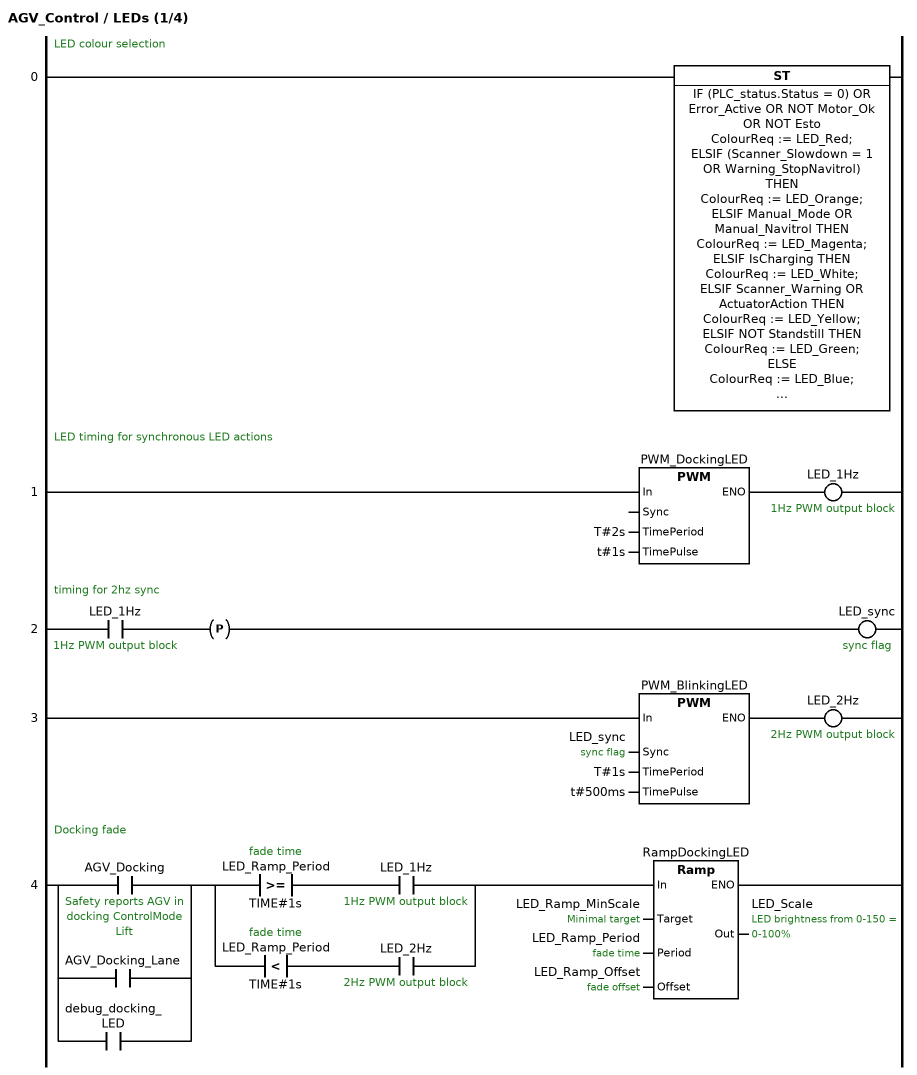
(* [picture p19: AGV_Control / LEDs, rungs 0-4] *)
(* Rung 0: LED colour selection *)
IF (PLC_status.Status = 0) OR Error_Active OR NOT Motor_Ok OR NOT Estop_Out OR (Warning_Mqtt_Client_Error AND InProd) THEN
	ColourReq := LED_Red;
ELSIF (Scanner_Slowdown = 1 OR Warning_StopNavitrol) THEN
	ColourReq := LED_Orange;
ELSIF Manual_Mode OR Manual_Navitrol THEN
	ColourReq := LED_Magenta;
ELSIF IsCharging THEN
	ColourReq := LED_White;
ELSIF Scanner_Warning OR ActuatorAction THEN
	ColourReq := LED_Yellow;
ELSIF NOT Standstill THEN
	ColourReq := LED_Green;
ELSE
	ColourReq := LED_Blue;
END_IF;

IF NOT debug_LED THEN
	Colour := ColourReq;
ELSE
	Colour := debug_Colour;
END_IF;

CASE Colour OF
	LED_Red:
		LED_R_Req := 100;
		LED_G_Req := 0;
		LED_B_Req := 0;
	LED_Orange:
		LED_R_Req := 100;
		LED_G_Req := 50;
		LED_B_Req := 0;
	LED_Yellow:
		LED_R_Req := 75;
		LED_G_Req := 75;
		LED_B_Req := 0;
	LED_Green:
		LED_R_Req := 0;
		LED_G_Req := 100;
		LED_B_Req := 0;
	LED_Cyan:
		LED_R_Req := 0;
		LED_G_Req := 100;
		LED_B_Req := 100;
	LED_Blue:
		LED_R_Req := 0;
		LED_G_Req := 0;
		LED_B_Req := 100;
	LED_Magenta:
		LED_R_Req := 100;
		LED_G_Req := 0;
		LED_B_Req := 100;
	LED_White:
		LED_R_Req := 100;
		LED_G_Req := 100;
		LED_B_Req := 100;
END_CASE;

IF (Colour = LED_Colour#LED_Orange) THEN
	LED_R := LED_R_Req*LED_Scale;
	LED_G := LED_G_Req*LED_Scale;//REAL_TO_INT(LED_R / 2) + ((LED_Ramp_Offset-LED_Scale) * 8);
	LED_B := LED_B_Req*LED_Scale;
ELSE
	LED_R := LED_R_Req*LED_Scale;
	LED_G := LED_G_Req*LED_Scale;
	LED_B := LED_B_Req*LED_Scale;
END_IF;

IF DomeLEDs THEN
	 if( LED_R>0) AND (Colour <> LED_Colour#LED_Orange) THEN 
		 IF NOT AGV_Docking THEN
		 	O_LED_R := TRUE; 
		ELSE 
			O_LED_R := LED_1Hz;
		END_IF;
	 ELSE
		 O_LED_R := FALSE;
	 END_IF;
	 
	 if( LED_G>0)  THEN 
		 IF NOT AGV_Docking THEN
		 	O_LED_G := TRUE; 
		ELSE 
			O_LED_G := LED_1Hz;
		END_IF;
	 ELSE
		 O_LED_G := FALSE;
	 END_IF;

	 if( LED_B>0) OR (Colour = LED_Colour#LED_Orange) THEN 
		 IF NOT AGV_Docking THEN
		 	O_LED_B := TRUE; 
		ELSE 
			O_LED_B := LED_1Hz;
		END_IF;
	 ELSE
		 O_LED_B := FALSE;
	 END_IF;
END_IF;

IF (LED_Scale < 0) THEN
	LED_Scale := 0;
END_IF;
IF IsCharging OR NOT (AGV_Docking OR debug_docking_LED) THEN
	LED_Scale:= LED_Ramp_Offset;
END_IF;

isCharging := Charge_Relay AND Navitrol_Battery.Voltage > 267;
(* Rung 1: LED timing for synchronous LED actions *)
PWM_DockingLED(In := TRUE, TimePeriod := T#2s, TimePulse := t#1s);
LED_1Hz := PWM_DockingLED.ENO;
(* Rung 2: timing for 2hz sync *)
_e36(CLK := LED_1Hz);
LED_sync := _e36.Q;
(* Rung 3 *)
PWM_BlinkingLED(In := TRUE, Sync := LED_sync, TimePeriod := T#1s, TimePulse := t#500ms);
LED_2Hz := PWM_BlinkingLED.ENO;
(* Rung 4: Docking fade *)
RampDockingLED(In := (AGV_Docking OR AGV_Docking_Lane OR debug_docking_LED) AND (((LED_Ramp_Period >= TIME#1s) AND LED_1Hz) OR ((LED_Ramp_Period < TIME#1s) AND LED_2Hz)), Target := LED_Ramp_MinScale, Period := LED_Ramp_Period, Offset := LED_Ramp_Offset, Out => LED_Scale);

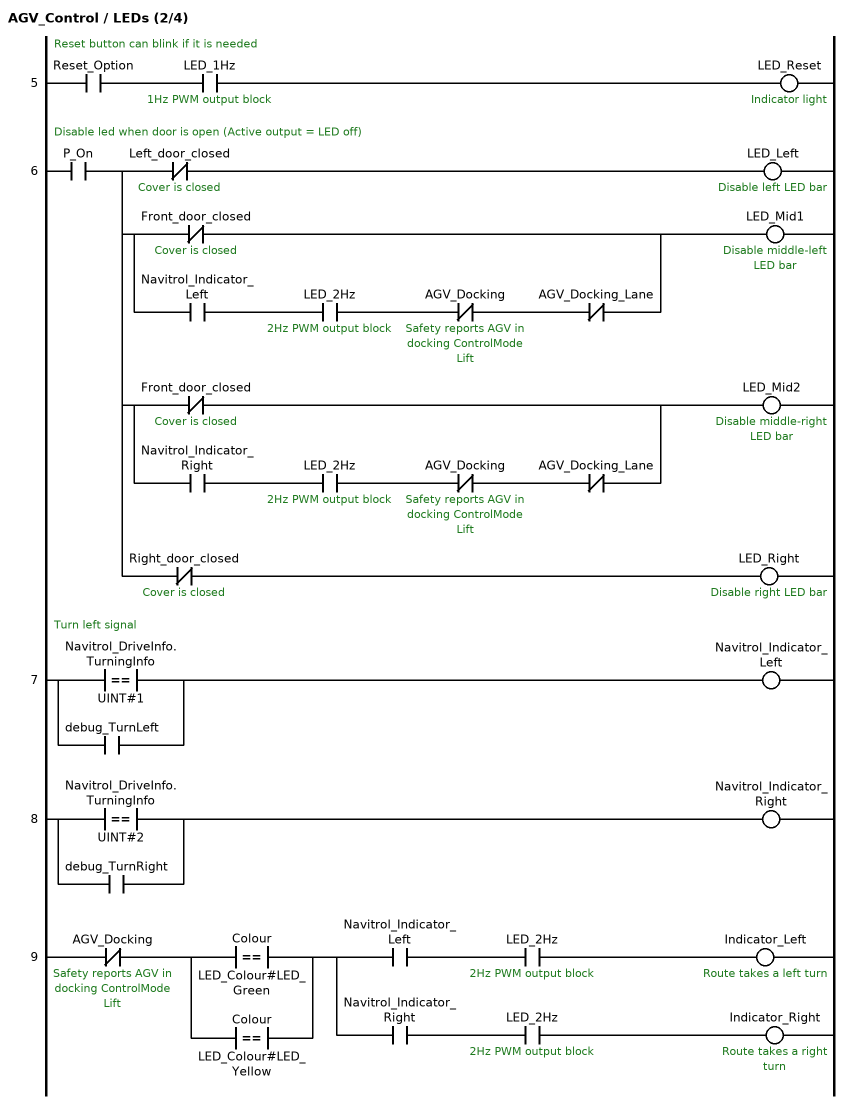
(* Rung 5: Reset button can blink if it is needed *)
LED_Reset := Reset_Option AND LED_1Hz;
(* Rung 6: Disable led when door is open (Active output = LED off) *)
LED_Left := P_On AND NOT Left_door_closed;
LED_Mid1 := P_On AND (NOT Front_door_closed OR (Navitrol_Indicator_Left AND LED_2Hz AND NOT AGV_Docking AND NOT AGV_Docking_Lane));
LED_Mid2 := P_On AND (NOT Front_door_closed OR (Navitrol_Indicator_Right AND LED_2Hz AND NOT AGV_Docking AND NOT AGV_Docking_Lane));
LED_Right := P_On AND NOT Right_door_closed;
(* Rung 7: Turn left signal *)
Navitrol_Indicator_Left := (Navitrol_DriveInfo.TurningInfo = UINT#1) OR debug_TurnLeft;
(* Rung 8 *)
Navitrol_Indicator_Right := (Navitrol_DriveInfo.TurningInfo = UINT#2) OR debug_TurnRight;
(* Rung 9 *)
_p37 := NOT AGV_Docking AND ((Colour = LED_Colour#LED_Green) OR (Colour = LED_Colour#LED_Yellow));
Indicator_Left := _p37 AND Navitrol_Indicator_Left AND LED_2Hz;
Indicator_Right := _p37 AND Navitrol_Indicator_Right AND LED_2Hz;

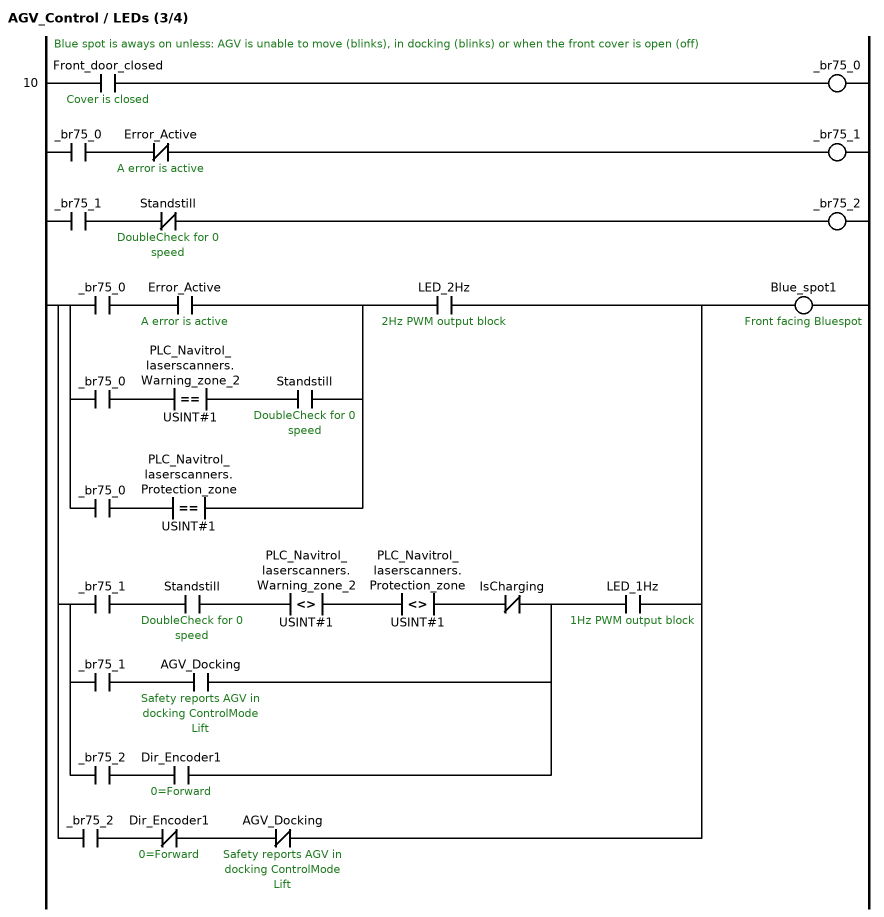
(* Rung 10: Blue spot is aways on unless: AGV is unable to move (blinks), in docking (blinks) or when the front cover is open (off) *)
_br75_0 := Front_door_closed;
_br75_1 := _br75_0 AND NOT Error_Active;
_br75_2 := _br75_1 AND NOT Standstill;
Blue_spot1 := (((_br75_0 AND Error_Active) OR (_br75_0 AND (PLC_Navitrol_laserscanners.Warning_zone_2 = USINT#1) AND Standstill) OR (_br75_0 AND (PLC_Navitrol_laserscanners.Protection_zone = USINT#1))) AND LED_2Hz) OR (((_br75_1 AND Standstill AND (PLC_Navitrol_laserscanners.Warning_zone_2 <> USINT#1) AND (PLC_Navitrol_laserscanners.Protection_zone <> USINT#1) AND NOT IsCharging) OR (_br75_1 AND AGV_Docking) OR (_br75_2 AND Dir_Encoder1)) AND LED_1Hz) OR (_br75_2 AND NOT Dir_Encoder1 AND NOT AGV_Docking);

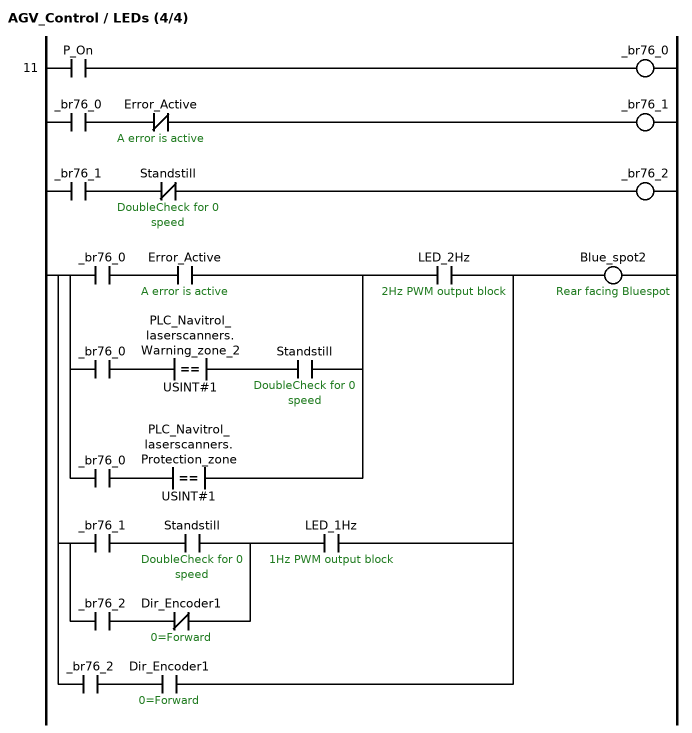
(* Rung 11 *)
_br76_0 := P_On;
_br76_1 := _br76_0 AND NOT Error_Active;
_br76_2 := _br76_1 AND NOT Standstill;
Blue_spot2 := (((_br76_0 AND Error_Active) OR (_br76_0 AND (PLC_Navitrol_laserscanners.Warning_zone_2 = USINT#1) AND Standstill) OR (_br76_0 AND (PLC_Navitrol_laserscanners.Protection_zone = USINT#1))) AND LED_2Hz) OR (((_br76_1 AND Standstill) OR (_br76_2 AND NOT Dir_Encoder1)) AND LED_1Hz) OR (_br76_2 AND Dir_Encoder1);

(* Section MES: ladder, written here as Structured Text *)

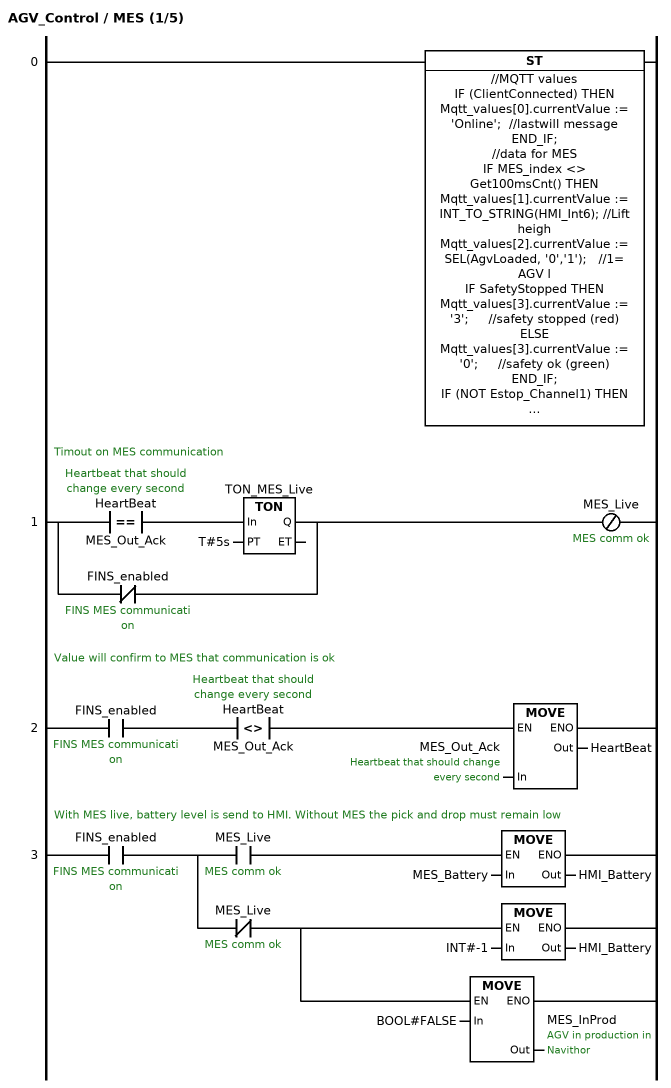
(* Rung 0 *)
//MQTT values
IF (ClientConnected) THEN
	Mqtt_values[0].currentValue := 'Online';	//lastwill message
END_IF;
//data for MES
IF MES_index <> Get100msCnt() THEN
	Mqtt_values[1].currentValue := INT_TO_STRING(HMI_Int6);	//Lift height in mm
	Mqtt_values[2].currentValue := SEL(AgvLoaded, '0','1');		//1= AGV loaded
	IF SafetyStopped THEN
	    Mqtt_values[3].currentValue := '3';			//safety stopped (red)
	ELSE
	    Mqtt_values[3].currentValue := '0';			//safety ok (green)
	END_IF;
	IF (NOT Estop_Channel1) THEN
		Mqtt_values[4].currentValue := '3';			//Estop button pressed (red)
	ELSIF (NOT Estop_Out) THEN
		Mqtt_values[4].currentValue := '2';			//Estop button ok, but not reset (yellow)
	ELSE
		Mqtt_values[4].currentValue := '0';			//Estop button ok (green)
	END_IF;
	Mqtt_values[5].currentValue := DINT_TO_STRING (EnumToNum(Scanner1_State));	//scanner status
	Mqtt_values[6].currentValue := DINT_TO_STRING (EnumToNum(Scanner2_State));	//scanner status
	Mqtt_values[7].currentValue := DINT_TO_STRING (EnumToNum(Scanner3_State));	//scanner status
	Mqtt_values[8].currentValue := SEL (OptionalFieldReq = 0,'1','0');	//1= Docking field active
	Mqtt_values[9].currentValue := SEL (Manual_Navitrol,'0','1');		//1= AGV in manualControlModeLift (navitrol)
	Mqtt_values[10].currentValue := SEL (HMI_Input5,'0','1');			//1= Lift in manual ControlModeLift
	Mqtt_values[11].currentValue := SEL (Brake_release,'0','1');	//1= Lift manually released
	Mqtt_values[12].currentValue := SEL (HMI_Int10 = 0,'0','1');	//1= AGV charging
	Mqtt_values[13].currentValue := SEL (MES_Request_Cancel, '0','1');	//1= MES can cancel order while AGV lowers fork
	IF (HMI_Int6 < 100 AND Mqtt_values[14].currentValue = '1' AND MES_Request_Cancel) OR Mqtt_values[14].currentValue = '' THEN
		Mqtt_values[14].currentValue := '0';	//order cancel completed, reset value
	END_IF;
	Mqtt_values[15].currentValue := SEL(Error_Fork_Object,'0','1');
	Mqtt_values[16].currentValue := INT_TO_STRING (CountedPallets);	//1= MES can cancel order while AGV lowers fork

	Mqtt_values[17].currentValue := SEL (lift_heavyLoad,'0','1');	//1 = There is heavy load on the forks
	Mqtt_values[18].currentValue := DINT_TO_STRING (EnumToNum(MES_LaneDropState)); // Lane drop state
	Mqtt_values[22].currentValue := SEL (HMI_Input11,'0','1');	//1= The question for certain action is answered with "Yes"
	Mqtt_values[23].currentValue := SEL (HMI_Input12,'0','1');	//1= The question for certain action is answered with "Cancel"
	Mqtt_values[24].currentValue := INT_TO_STRING(MES_Language);
	Mqtt_values[25].currentValue := DINT_TO_STRING (EnumToNum(MES_LanePickState)); // Lane drop state
	
	Navitrol_TargetDetectionStatusToMES.TargetFount := SEL	(Navitrol_TargetDetectionStatus.TargetFount= 01, '0,','1,'); 
	Navitrol_TargetDetectionStatusToMES.TargetReached := SEL	(Navitrol_TargetDetectionStatus.TargetReached= 01, '0,','1,'); 	
	Navitrol_TargetDetectionStatusToMES.TargetWithinSafetyDistance := SEL  (Navitrol_TargetDetectionStatus.TargetWithinSafetyDistance = 01, '0,','1,'); 	
	Navitrol_TargetDetectionStatusToMES.TargetX := 	(INT_TO_STRING (REAL_TO_INT (Navitrol_TargetDetectionStatus.TargetX*100 ))); 
	Navitrol_TargetDetectionStatusToMES.TargetY := (INT_TO_STRING (REAL_TO_INT 	(Navitrol_TargetDetectionStatus.TargetY*100))); 	
	Navitrol_TargetDetectionStatusToMES.Angle:= (INT_TO_STRING (REAL_TO_INT 	(Navitrol_TargetDetectionStatus.TargetAngle*100))); 
	
	Mqtt_values[19].currentValue :=CONCAT (Navitrol_TargetDetectionStatusToMES.TargetFount,Navitrol_TargetDetectionStatusToMES.TargetReached,
	Navitrol_TargetDetectionStatusToMES.TargetWithinSafetyDistance,CONCAT (Navitrol_TargetDetectionStatusToMES.TargetX,','),Navitrol_TargetDetectionStatusToMES.TargetY);

	Mqtt_values[21].currentValue :=Navitrol_TargetDetectionStatusToMES.Angle;
	//error list to MES
	IF Navitrol_ErrorWithLevel.ErrorCount = 0 THEN
		//no error, clear values
		Mqtt_values[20].currentValue := '';
	ELSE
		ErrorString := '';
		FOR index := 0 TO UDINT_TO_INT(Navitrol_ErrorWithLevel.ErrorCount)-1 DO
			ErrorString := CONCAT(ErrorString, UDINT_TO_STRING(Navitrol_ErrorWithLevel.ErrorList[index].ErrorCode),',');
		END_FOR;
		Mqtt_values[20].currentValue := ErrorString;
	END_IF;
	
	MES_index := Get100msCnt();
END_IF;
//MQTT actuator request
(* Rung 1: Timout on MES communication *)
TON_MES_Live(In := HeartBeat = MES_Out_Ack, PT := T#5s);
MES_Live := NOT (TON_MES_Live.Q OR NOT FINS_enabled);
(* Rung 2: Value will confirm to MES that communication is ok *)
IF FINS_enabled AND (HeartBeat <> MES_Out_Ack) THEN HeartBeat := MES_Out_Ack; END_IF;
(* Rung 3: With MES live, battery level is send to HMI. Without MES the pick and drop must remain low *)
IF FINS_enabled AND MES_Live THEN HMI_Battery := MES_Battery; END_IF;
IF FINS_enabled AND NOT MES_Live THEN
    HMI_Battery := INT#-1;
    MES_InProd := BOOL#FALSE;
END_IF;

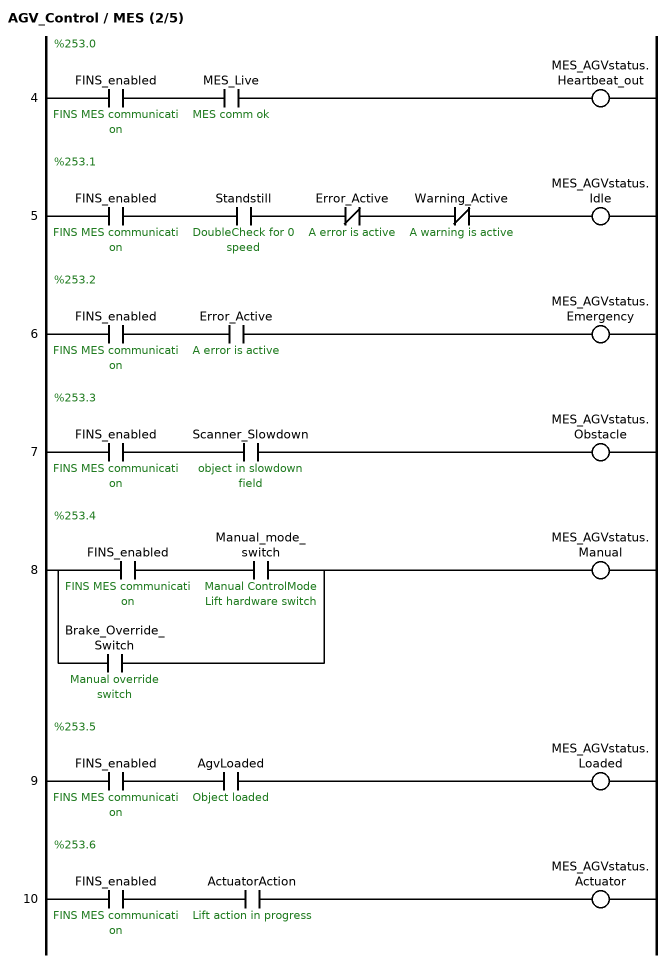
(* Rung 4: %253.0 *)
MES_AGVstatus.Heartbeat_out := FINS_enabled AND MES_Live;
(* Rung 5: %253.1 *)
MES_AGVstatus.Idle := FINS_enabled AND Standstill AND NOT Error_Active AND NOT Warning_Active;
(* Rung 6: %253.2 *)
MES_AGVstatus.Emergency := FINS_enabled AND Error_Active;
(* Rung 7: %253.3 *)
MES_AGVstatus.Obstacle := FINS_enabled AND Scanner_Slowdown;
(* Rung 8: %253.4 *)
MES_AGVstatus.Manual := (FINS_enabled AND Manual_mode_switch) OR Brake_Override_Switch;
(* Rung 9: %253.5 *)
MES_AGVstatus.Loaded := FINS_enabled AND AgvLoaded;
(* Rung 10: %253.6 *)
MES_AGVstatus.Actuator := FINS_enabled AND ActuatorAction;

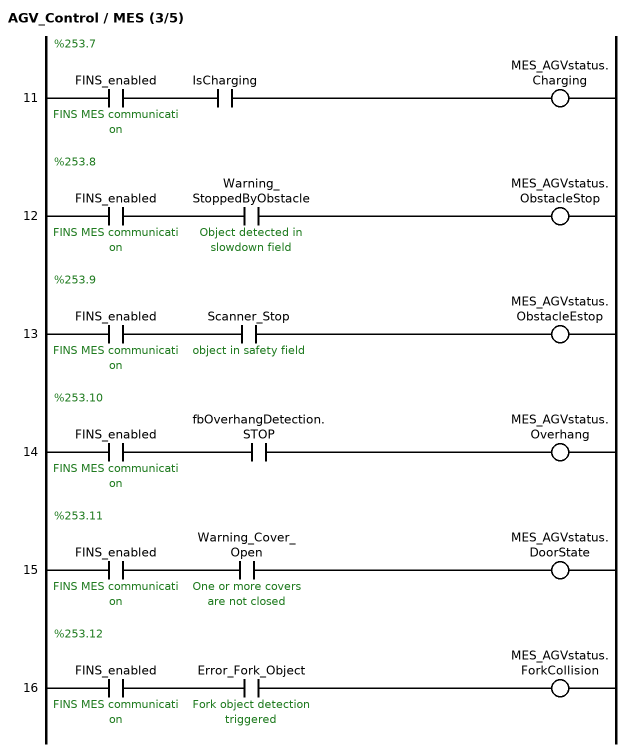
(* Rung 11: %253.7 *)
MES_AGVstatus.Charging := FINS_enabled AND IsCharging;
(* Rung 12: %253.8 *)
MES_AGVstatus.ObstacleStop := FINS_enabled AND Warning_StoppedByObstacle;
(* Rung 13: %253.9 *)
MES_AGVstatus.ObstacleEstop := FINS_enabled AND Scanner_Stop;
(* Rung 14: %253.10 *)
MES_AGVstatus.Overhang := FINS_enabled AND fbOverhangDetection.STOP;
(* Rung 15: %253.11 *)
MES_AGVstatus.DoorState := FINS_enabled AND Warning_Cover_Open;
(* Rung 16: %253.12 *)
MES_AGVstatus.ForkCollision := FINS_enabled AND Error_Fork_Object;

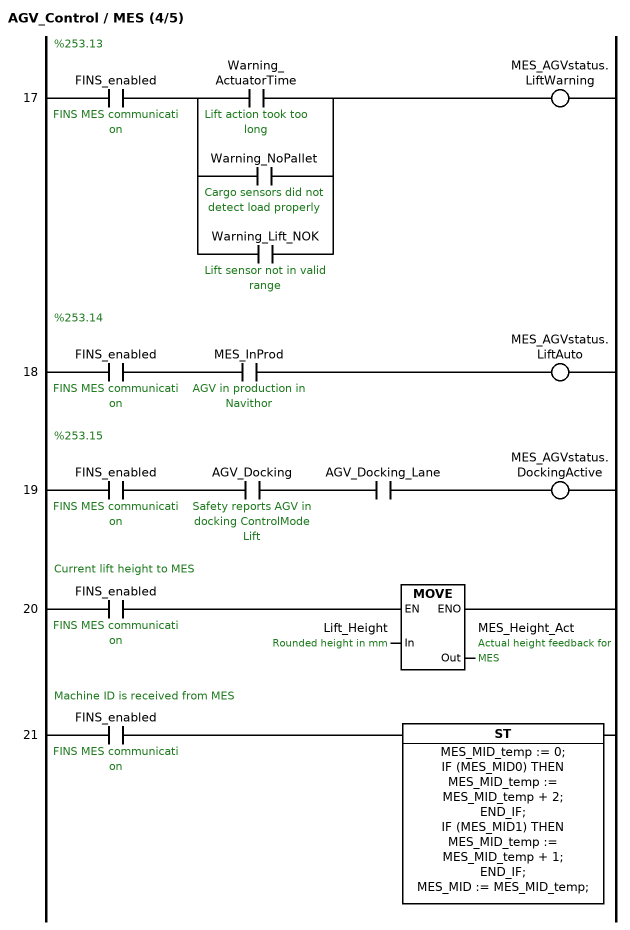
(* Rung 17: %253.13 *)
MES_AGVstatus.LiftWarning := FINS_enabled AND (Warning_ActuatorTime OR Warning_NoPallet OR Warning_Lift_NOK);
(* Rung 18: %253.14 *)
MES_AGVstatus.LiftAuto := FINS_enabled AND MES_InProd;
(* Rung 19: %253.15 *)
MES_AGVstatus.DockingActive := FINS_enabled AND AGV_Docking AND AGV_Docking_Lane;
(* Rung 20: Current lift height to MES *)
IF FINS_enabled THEN MES_Height_Act := Lift_Height; END_IF;
(* Rung 21: Machine ID is received from MES *)
IF FINS_enabled THEN
    MES_MID_temp := 0;
    IF (MES_MID0) THEN
    	MES_MID_temp := MES_MID_temp + 2;
    END_IF;
    IF (MES_MID1) THEN
    	MES_MID_temp := MES_MID_temp + 1;
    END_IF;
    MES_MID := MES_MID_temp;
END_IF;

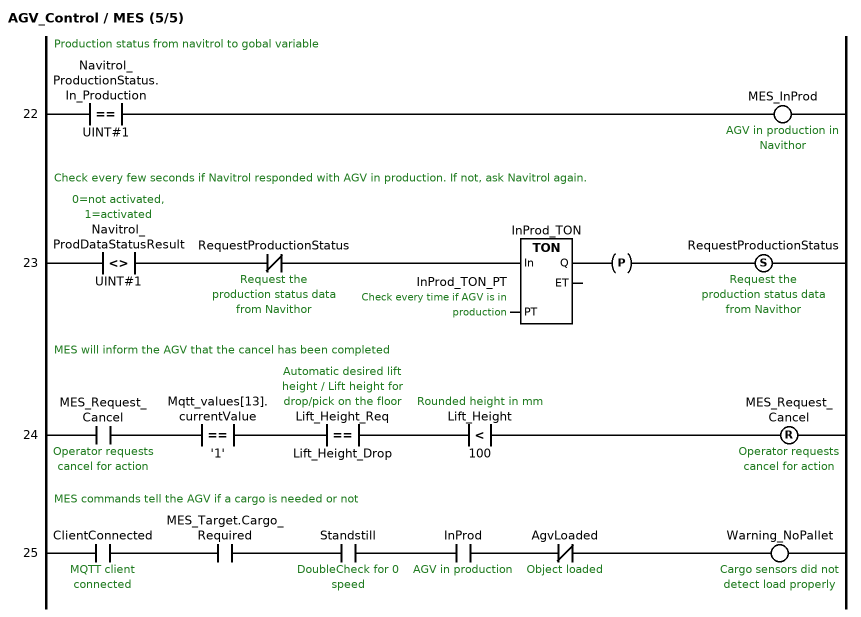
(* Rung 22: Production status from navitrol to gobal variable *)
MES_InProd := Navitrol_ProductionStatus.In_Production = UINT#1;
(* Rung 23: Check every few seconds if Navitrol responded with AGV in production. If not, ask Navitrol again. *)
InProd_TON(In := (Navitrol_ProdDataStatusResult <> UINT#1) AND NOT RequestProductionStatus, PT := InProd_TON_PT);
_e38(CLK := InProd_TON.Q);
IF _e38.Q THEN RequestProductionStatus := TRUE; END_IF;
(* Rung 24: MES will inform the AGV that the cancel has been completed *)
IF MES_Request_Cancel AND (Mqtt_values[13].currentValue = '1') AND (Lift_Height_Req = Lift_Height_Drop) AND (Lift_Height < 100) THEN
    MES_Request_Cancel := FALSE;
END_IF;
(* Rung 25: MES commands tell the AGV if a cargo is needed or not *)
Warning_NoPallet := ClientConnected AND MES_Target.Cargo_Required AND Standstill AND InProd AND NOT AgvLoaded;

(* Section HMI: ladder, written here as Structured Text *)

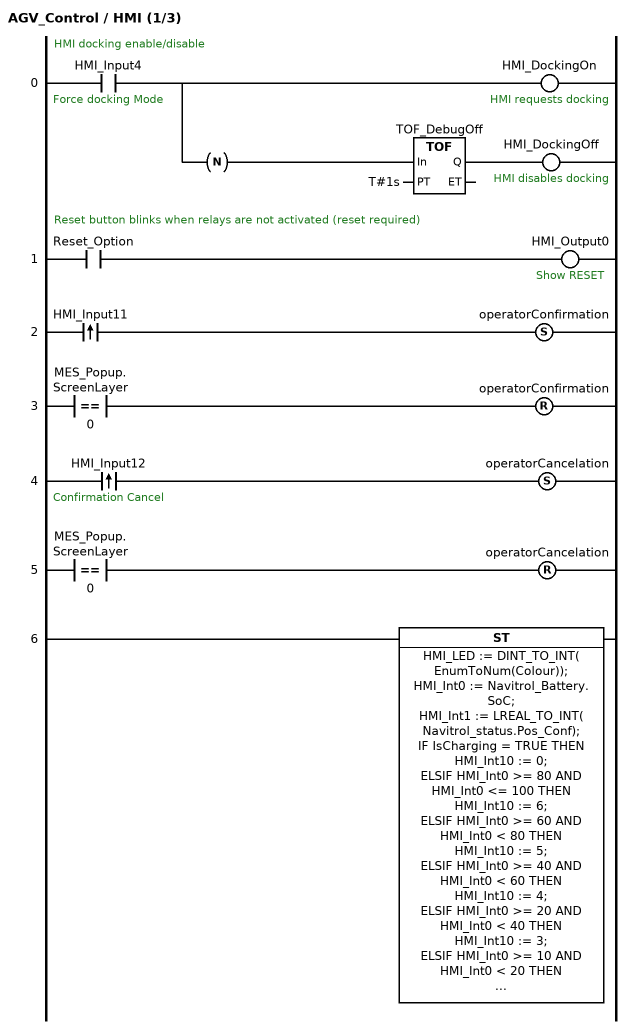
(* Rung 0: HMI docking enable/disable *)
HMI_DockingOn := HMI_Input4;
_e39(CLK := HMI_Input4);
TOF_DebugOff(In := _e39.Q, PT := T#1s);
HMI_DockingOff := TOF_DebugOff.Q;
(* Rung 1: Reset button blinks when relays are not activated (reset required) *)
HMI_Output0 := Reset_Option;
(* Rung 2 *)
_e40(CLK := HMI_Input11);
IF _e40.Q THEN operatorConfirmation := TRUE; END_IF;
(* Rung 3 *)
IF MES_Popup.ScreenLayer = 0 THEN operatorConfirmation := FALSE; END_IF;
(* Rung 4 *)
_e41(CLK := HMI_Input12);
IF _e41.Q THEN operatorCancelation := TRUE; END_IF;
(* Rung 5 *)
IF MES_Popup.ScreenLayer = 0 THEN operatorCancelation := FALSE; END_IF;
(* Rung 6 *)
HMI_LED := DINT_TO_INT(EnumToNum(Colour));

HMI_Int0 := Navitrol_Battery.SoC;
HMI_Int1 := LREAL_TO_INT(Navitrol_status.Pos_Conf);

IF IsCharging = TRUE THEN
	HMI_Int10 := 0;
ELSIF HMI_Int0 >= 80 AND HMI_Int0 <= 100 THEN
	HMI_Int10 := 6;
ELSIF HMI_Int0 >= 60 AND HMI_Int0 < 80 THEN
	HMI_Int10 := 5;
ELSIF HMI_Int0 >= 40 AND HMI_Int0 < 60 THEN
	HMI_Int10 := 4;
ELSIF HMI_Int0 >= 20 AND HMI_Int0 < 40 THEN
	HMI_Int10 := 3;
ELSIF HMI_Int0 >= 10 AND HMI_Int0 < 20 THEN
	HMI_Int10 := 2;
ELSE  //HMI_Int0 < 10 & not charging
	HMI_Int10 := 1;
END_IF;

//front scanners cmbined till HMI is updated
IF NOT Scan1_Stop OR NOT Scan2_Stop THEN
	Scanner1_State := State_Scanner#SCAN_eStop;
	Scanner2_State := State_Scanner#SCAN_eStop;
	HMI_Int2 := 0;
ELSIF NOT Scan1_Slow OR NOT Scan2_Slow THEN
	Scanner1_State := State_Scanner#SCAN_Stop;
	Scanner2_State := State_Scanner#SCAN_Stop;
	HMI_Int2 := 3;
ELSIF NOT Scan1_Warn OR NOT Scan2_Warn THEN
	Scanner1_State := State_Scanner#SCAN_Warn;
	Scanner2_State := State_Scanner#SCAN_Warn;
	HMI_Int2 := 2;
ELSE
	Scanner1_State := State_Scanner#SCAN_Clear;
	Scanner2_State := State_Scanner#SCAN_Clear;
	HMI_Int2:= 1;
END_IF;

//Fork scanner
IF NOT Scan3_Stop  AND NOT ( OptionalFieldReq =1 OR OptionalFieldReq= 2) THEN
	Scanner2_State := State_Scanner#SCAN_eStop;
	HMI_Int3 := 0;
ELSIF NOT Scan3_slow AND NOT ( OptionalFieldReq =1 OR OptionalFieldReq= 2) THEN
	Scanner2_State := State_Scanner#SCAN_Stop;
	HMI_Int3 := 3;
ELSIF NOT Scan3_Warn  AND  NOT ( OptionalFieldReq =1 OR OptionalFieldReq= 2) THEN
	Scanner2_State := State_Scanner#SCAN_Warn;
	HMI_Int3 := 2;
ELSE
	Scanner2_State := State_Scanner#SCAN_Clear;
	HMI_Int3:= 1;
END_IF;

IF NOT Estop_Out THEN
	IF (Estop_Channel1 AND RM_Estop) THEN
		HMI_Int4 := 2;
	ELSE
		HMI_Int4 := 0;
	END_IF;
ELSE
	HMI_Int4 := 1;
END_IF;

HMI_Int5 := MachineID;
HMI_Int6 := Lift_Height;

HMI_Int8 := LiftHeightMin;
HMI_Int9 := LiftHeightMax;

// Activation of popup interaction with operator
HMI_Int11:=MES_Popup.ScreenLayer;
HMI_String1 := MES_Popup.Message;

MES_Language := HMI_Int16;

MES_Language := HMI_Int16;

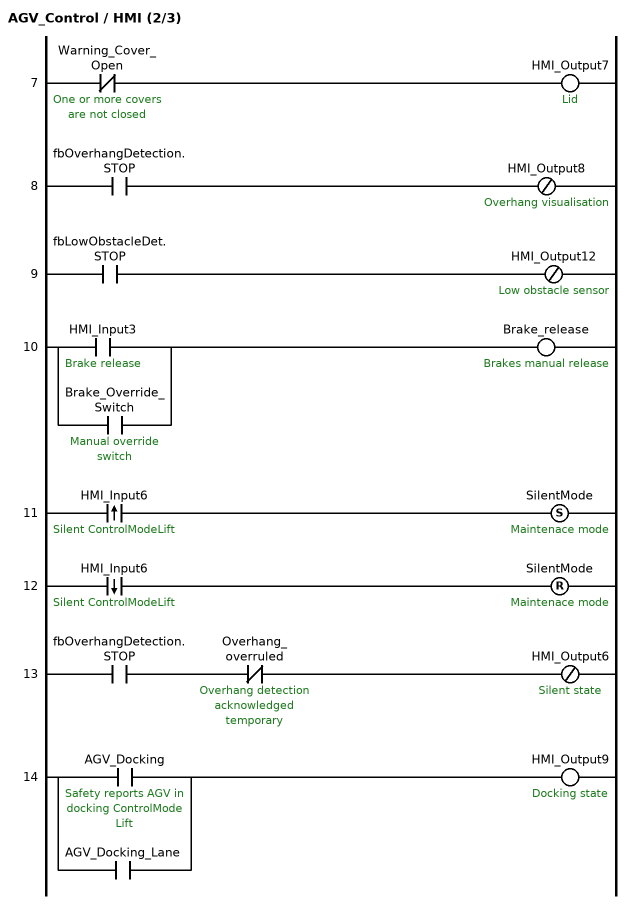
(* Rung 7 *)
HMI_Output7 := NOT Warning_Cover_Open;
(* Rung 8 *)
HMI_Output8 := NOT fbOverhangDetection.STOP;
(* Rung 9 *)
HMI_Output12 := NOT fbLowObstacleDet.STOP;
(* Rung 10 *)
Brake_release := HMI_Input3 OR Brake_Override_Switch;
(* Rung 11 *)
_e42(CLK := HMI_Input6);
IF _e42.Q THEN SilentMode := TRUE; END_IF;
(* Rung 12 *)
_e43(CLK := HMI_Input6);
IF _e43.Q THEN SilentMode := FALSE; END_IF;
(* Rung 13 *)
HMI_Output6 := NOT (fbOverhangDetection.STOP AND NOT Overhang_overruled);
(* Rung 14 *)
HMI_Output9 := AGV_Docking OR AGV_Docking_Lane;

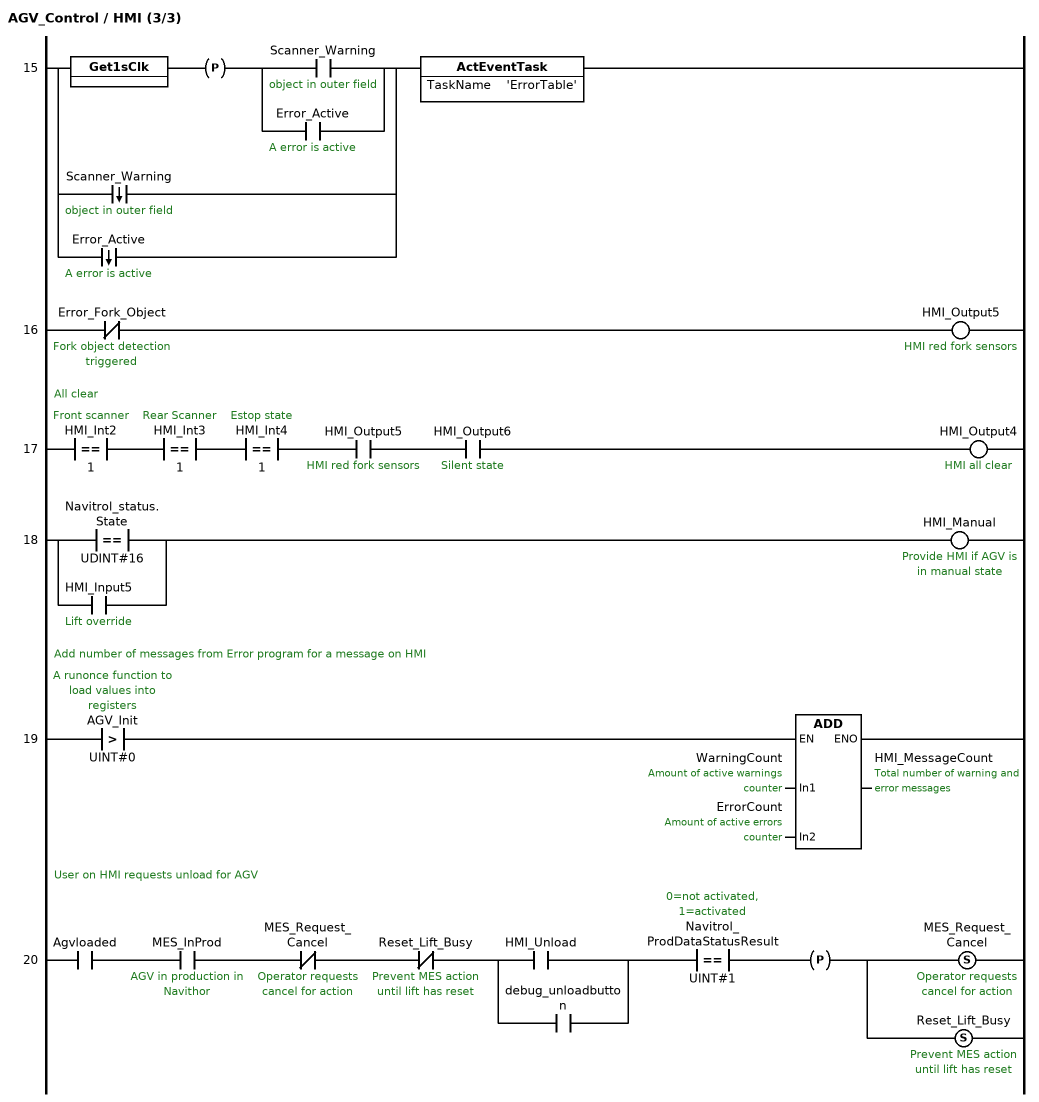
(* Rung 15 *)
_e44(CLK := Get1sClk());
_e45(CLK := Scanner_Warning);
_e46(CLK := Error_Active);
(* drawn but driving nothing: 'ErrorTable' *)
(* Rung 16 *)
HMI_Output5 := NOT Error_Fork_Object;
(* Rung 17: All clear *)
HMI_Output4 := (HMI_Int2 = 1) AND (HMI_Int3 = 1) AND (HMI_Int4 = 1) AND HMI_Output5 AND HMI_Output6;
(* Rung 18 *)
HMI_Manual := (Navitrol_status.State = UDINT#16) OR HMI_Input5;
(* Rung 19: Add number of messages from Error program for a message on HMI *)
IF AGV_Init > UINT#0 THEN HMI_MessageCount := WarningCount + ErrorCount; END_IF;
(* Rung 20: User on HMI requests unload for AGV *)
_e47(CLK := Agvloaded AND MES_InProd AND NOT MES_Request_Cancel AND NOT Reset_Lift_Busy AND (HMI_Unload OR debug_unloadbutton) AND (Navitrol_ProdDataStatusResult = UINT#1));
IF _e47.Q THEN
    MES_Request_Cancel := TRUE;
    Reset_Lift_Busy := TRUE;
END_IF;

(* Section Error: ladder, written here as Structured Text *)

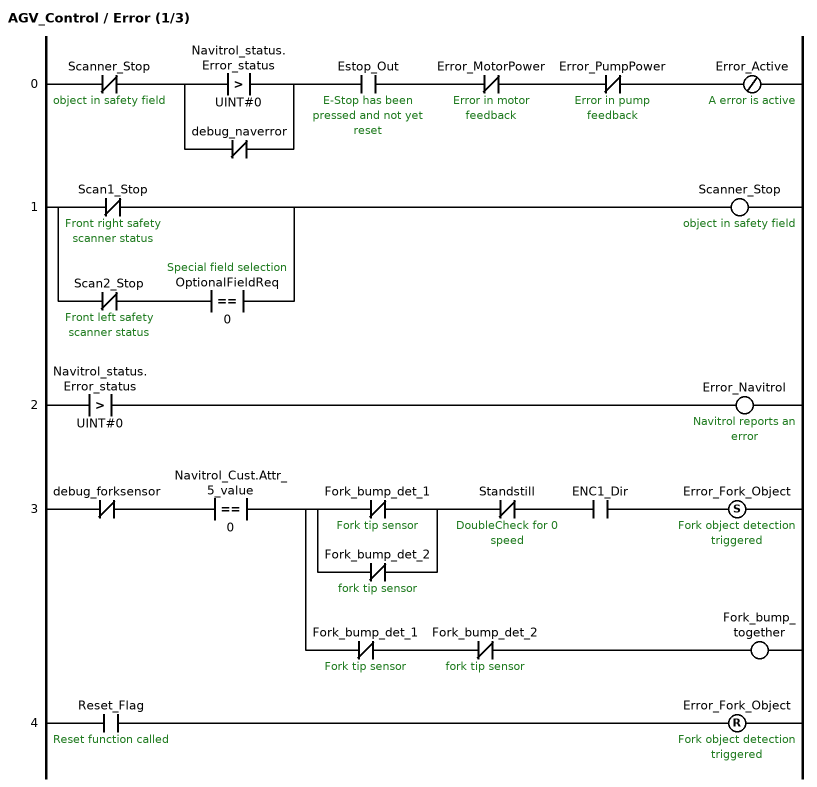
(* Rung 0 *)
Error_Active := NOT (NOT Scanner_Stop AND ((Navitrol_status.Error_status > UINT#0) OR NOT debug_naverror) AND Estop_Out AND NOT Error_MotorPower AND NOT Error_PumpPower);
(* Rung 1 *)
Scanner_Stop := NOT Scan1_Stop OR (NOT Scan2_Stop AND (OptionalFieldReq = 0));
(* Rung 2 *)
Error_Navitrol := Navitrol_status.Error_status > UINT#0;
(* Rung 3 *)
_p48 := NOT debug_forksensor AND (Navitrol_Cust.Attr_5_value = 0);
IF _p48 AND (NOT Fork_bump_det_1 OR NOT Fork_bump_det_2) AND NOT Standstill AND ENC1_Dir THEN
    Error_Fork_Object := TRUE;
END_IF;
Fork_bump_together := _p48 AND NOT Fork_bump_det_1 AND NOT Fork_bump_det_2;
(* Rung 4 *)
IF Reset_Flag THEN Error_Fork_Object := FALSE; END_IF;

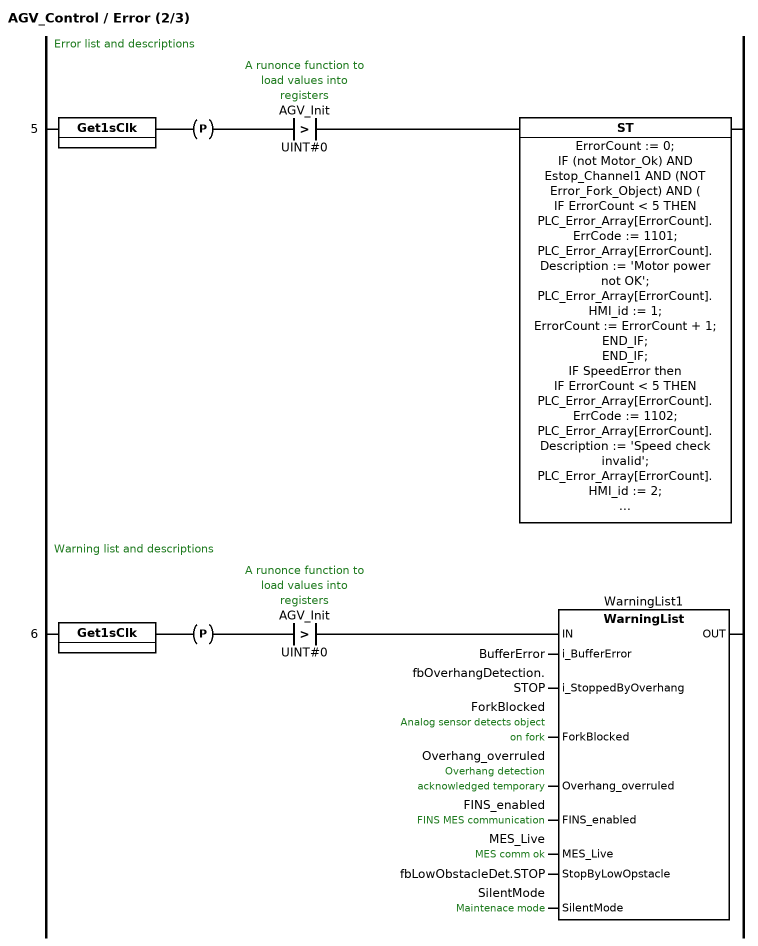
(* Rung 5: Error list and descriptions *)
_e49(CLK := Get1sClk());
IF _e49.Q AND (AGV_Init > UINT#0) THEN
    ErrorCount := 0;
    
    IF (not Motor_Ok) AND Estop_Channel1 AND (NOT Error_Fork_Object) AND (NOT Docking_error) then
    	IF ErrorCount < 5 THEN
    		PLC_Error_Array[ErrorCount].ErrCode := 1101;
    		PLC_Error_Array[ErrorCount].Description := 'Motor power not OK';
    		PLC_Error_Array[ErrorCount].HMI_id := 1;
    		ErrorCount := ErrorCount + 1;
    	END_IF;
    END_IF;
    
    IF SpeedError then
    	IF ErrorCount < 5 THEN
    		PLC_Error_Array[ErrorCount].ErrCode := 1102;
    		PLC_Error_Array[ErrorCount].Description := 'Speed check invalid';
    		PLC_Error_Array[ErrorCount].HMI_id := 2;
    		ErrorCount := ErrorCount + 1;
    	END_IF;
    END_IF;
    
    IF (not Pump_Ok) AND Estop_Out AND (NOT Error_Fork_Object) then
    	IF ErrorCount < 5 THEN
    		PLC_Error_Array[ErrorCount].ErrCode := 1201;
    		PLC_Error_Array[ErrorCount].Description := 'Lift power not OK';
    		PLC_Error_Array[ErrorCount].HMI_id := 3;
    		ErrorCount := ErrorCount + 1;
    	END_IF;
    END_IF;
    IF heavyLoad.Q1 THEN
    	IF ErrorCount < 5 THEN
    		PLC_Error_Array[ErrorCount].ErrCode := 1202;
    		PLC_Error_Array[ErrorCount].Description := 'Heavy load, max hight';
    		PLC_Error_Array[ErrorCount].HMI_id := 15;
    		ErrorCount := ErrorCount + 1;
    	END_IF;
    END_IF;
    
    //IF Error_Navitrol then
    //	IF ErrorCount < 5 THEN
    //		PLC_Error_Array[ErrorCount].ErrCode := 1301;
    //		PLC_Error_Array[ErrorCount].Description := 'ERR_NAVITROL_TO_PLC';
    //		ErrorCount := ErrorCount + 1;
    //	END_IF;
    //END_IF;
    
    IF (NOT Estop_Channel1 & NOT Estop_Out) THEN
    	IF ErrorCount < 5 THEN
    		PLC_Error_Array[ErrorCount].ErrCode := 1401;
    		PLC_Error_Array[ErrorCount].Description := 'E-stop button pressed';
    		PLC_Error_Array[ErrorCount].HMI_id := 4;
    		ErrorCount := ErrorCount + 1;
    	END_IF;
    END_IF;
    
    IF (Estop_Channel1 & NOT Estop_Out) THEN
    	IF ErrorCount < 5 THEN
    		PLC_Error_Array[ErrorCount].ErrCode := 1402;
    		PLC_Error_Array[ErrorCount].Description := 'E-stop reset required';
    		PLC_Error_Array[ErrorCount].HMI_id := 5;
    		ErrorCount := ErrorCount + 1;
    	END_IF;
    END_IF;
    
    IF (Scanner_Warning & Scanner_Slowdown & Scanner_Stop) THEN
    	IF ErrorCount < 5 THEN
    		PLC_Error_Array[ErrorCount].ErrCode := 1403;
    		PLC_Error_Array[ErrorCount].Description := 'Object in safety field';
    		PLC_Error_Array[ErrorCount].HMI_id := 6;
    		ErrorCount := ErrorCount + 1;
    	END_IF;
    END_IF;
    
    IF (NOT Scanner_Warning & NOT Scanner_Slowdown & Scanner_Stop) THEN
    	IF ErrorCount < 5 THEN
    		PLC_Error_Array[ErrorCount].ErrCode := 1404;
    		PLC_Error_Array[ErrorCount].Description := 'Scanner in fault';
    		PLC_Error_Array[ErrorCount].HMI_id := 7;
    		ErrorCount := ErrorCount + 1;
    	END_IF;
    END_IF;
    
    IF (Error_Fork_Object) THEN
    	IF ErrorCount < 5 THEN
    		PLC_Error_Array[ErrorCount].ErrCode := 1502;
    		PLC_Error_Array[ErrorCount].Description := 'Fork collision';
    		PLC_Error_Array[ErrorCount].HMI_id := 8;
    		ErrorCount := ErrorCount + 1;
    	END_IF;
    END_IF;
    
    IF (Docking_error) THEN
    	IF ErrorCount < 5 THEN
    		PLC_Error_Array[ErrorCount].ErrCode := 1503;
    		PLC_Error_Array[ErrorCount].Description := 'Docking error lane drop';
    		PLC_Error_Array[ErrorCount].HMI_id := 9;
    		ErrorCount := ErrorCount + 1;
    	END_IF;
    END_IF;
    IF (WarningCargoDrag) THEN
    	IF ErrorCount < 5 THEN
    		PLC_Error_Array[ErrorCount].ErrCode := 1504;
    		PLC_Error_Array[ErrorCount].Description := 'Cargo unload failure';
    		PLC_Error_Array[ErrorCount].HMI_id := 13;
    		ErrorCount := ErrorCount + 1;
    	END_IF;
    END_IF;
    
    IF NearTarget_No_Load = TRUE AND MES_Target.Cargo_Required = TRUE then
    	IF (ErrorCount < 5) THEN
    		PLC_Error_Array[4].ErrCode := 1505;
    		PLC_Error_Array[4].Description := 'Cargo load failure';
    		PLC_Error_Array[4].HMI_id := 13;
    	END_IF;
    END_IF;
    IF (ErrorCount < 4) THEN
    	PLC_Error_Array[3].ErrCode := 0;
    	PLC_Error_Array[3].Description := '                        ';
    	PLC_Error_Array[3].HMI_id := 0;
    END_IF;
    IF (ErrorCount < 3) THEN
    	PLC_Error_Array[2].ErrCode := 0;
    	PLC_Error_Array[2].Description := '                        ';
    	PLC_Error_Array[2].HMI_id := 0;
    END_IF;
    IF (ErrorCount < 2) THEN
    	PLC_Error_Array[1].ErrCode := 0;
    	PLC_Error_Array[1].Description := '                        ';
    	PLC_Error_Array[1].HMI_id := 0;
    END_IF;
    IF (ErrorCount < 1) THEN
    	//No active errors
    	PLC_Error_Array[0].ErrCode := 0;
    	PLC_Error_Array[0].Description := '                        ';
    	PLC_Error_Array[0].HMI_id := 0;
    END_IF;
    
    //Handle the error strings
    FOR ErrorIndex := 0 to 4 DO
    	PLC_Error_Array[ErrorIndex].ActualChars := uint_to_byte(LEN(PLC_Error_Array[ErrorIndex].Description));
    	PLC_Error_Array[ErrorIndex].ZeroFill := int_to_byte(BYTE_TO_INT(PLC_Error_Array[ErrorIndex].DescrLength) -BYTE_TO_INT(PLC_Error_Array[ErrorIndex].ActualChars));
    END_FOR;
    
    //HMI_ErrorText1 := '                        ';
    //HMI_ErrorText2 := '                        ';
    //HMI_ErrorText3 := '                        ';
    //HMI_ErrorText4 := '                        ';
    //HMI_ErrorText5 := '                        ';
    
    HMI_Error1 := PLC_Error_Array[0].ErrCode;
    HMI_ErrorText1 := BYTE_TO_INT(PLC_Error_Array[0].HMI_id);
    HMI_Error2 := PLC_Error_Array[1].ErrCode;
    HMI_ErrorText2 := BYTE_TO_INT(PLC_Error_Array[1].HMI_id);
    HMI_Error3 := PLC_Error_Array[2].ErrCode;
    HMI_ErrorText3 := BYTE_TO_INT(PLC_Error_Array[2].HMI_id);
    HMI_Error4 := PLC_Error_Array[3].ErrCode;
    HMI_ErrorText4 := BYTE_TO_INT(PLC_Error_Array[3].HMI_id);
    HMI_Error5 := PLC_Error_Array[4].ErrCode;
    HMI_ErrorText5 := BYTE_TO_INT(PLC_Error_Array[4].HMI_id);
END_IF;
(* Rung 6: Warning list and descriptions *)
_e50(CLK := Get1sClk());
WarningList1(IN := _e50.Q AND (AGV_Init > UINT#0), i_BufferError := BufferError, i_StoppedByOverhang := fbOverhangDetection.STOP, ForkBlocked := ForkBlocked, Overhang_overruled := Overhang_overruled, FINS_enabled := FINS_enabled, MES_Live := MES_Live, StopByLowOpstacle := fbLowObstacleDet.STOP, SilentMode := SilentMode);

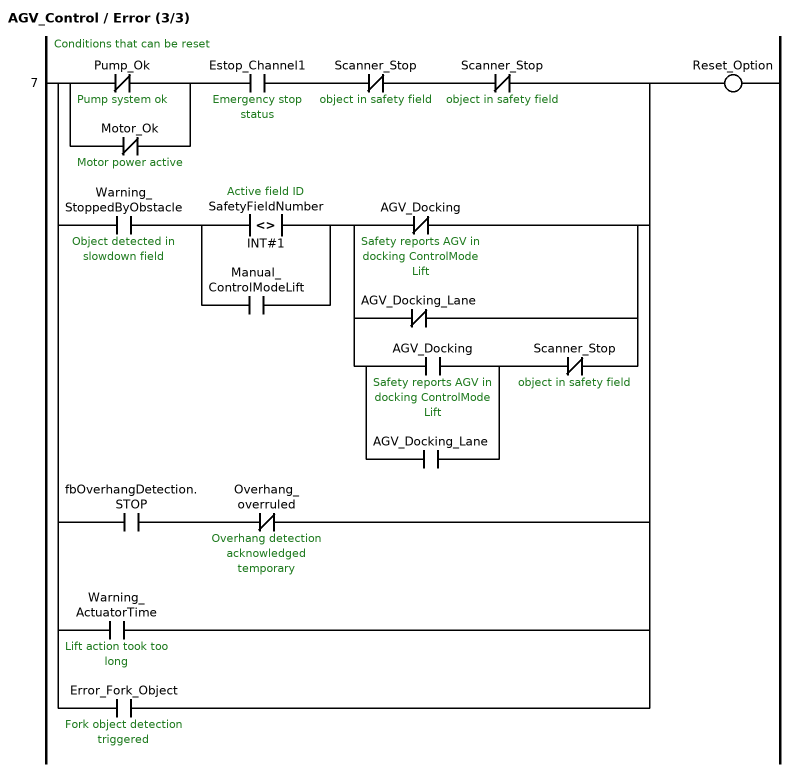
(* Rung 7: Conditions that can be reset *)
Reset_Option := ((NOT Pump_Ok OR NOT Motor_Ok) AND Estop_Channel1 AND NOT Scanner_Stop AND NOT Scanner_Stop) OR (Warning_StoppedByObstacle AND ((SafetyFieldNumber <> INT#1) OR Manual_ControlModeLift) AND (NOT AGV_Docking OR NOT AGV_Docking_Lane OR ((AGV_Docking OR AGV_Docking_Lane) AND NOT Scanner_Stop))) OR (fbOverhangDetection.STOP AND NOT Overhang_overruled) OR Warning_ActuatorTime OR Error_Fork_Object;

(* Section PalletDetecton: ladder, written here as Structured Text *)

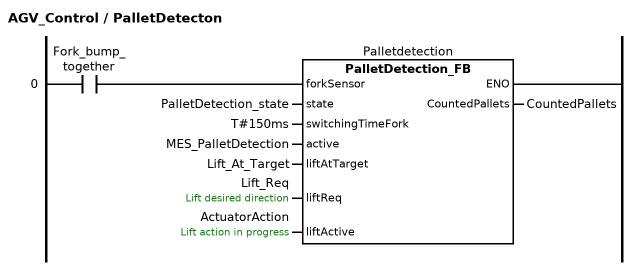
(* Rung 0 *)
Palletdetection(forkSensor := Fork_bump_together, state := PalletDetection_state, switchingTimeFork := T#150ms, active := MES_PalletDetection, liftAtTarget := Lift_At_Target, liftReq := Lift_Req, liftActive := ActuatorAction, CountedPallets => CountedPallets);

(* Section Overhang: ladder, written here as Structured Text *)

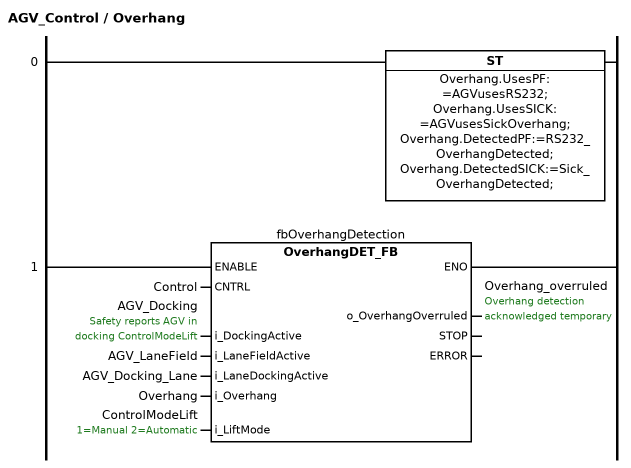
(* Rung 0 *)
Overhang.UsesPF:=AGVusesRS232;
Overhang.UsesSICK:=AGVusesSickOverhang;
Overhang.DetectedPF:=RS232_OverhangDetected;
Overhang.DetectedSICK:=Sick_OverhangDetected;
(* Rung 1 *)
fbOverhangDetection(ENABLE := TRUE, CNTRL := Control, i_DockingActive := AGV_Docking, i_LaneFieldActive := AGV_LaneField, i_LaneDockingActive := AGV_Docking_Lane, i_Overhang := Overhang, i_LiftMode := ControlModeLift, o_OverhangOverruled => Overhang_overruled);

(* Section LowObstacleDetection: ladder, written here as Structured Text *)

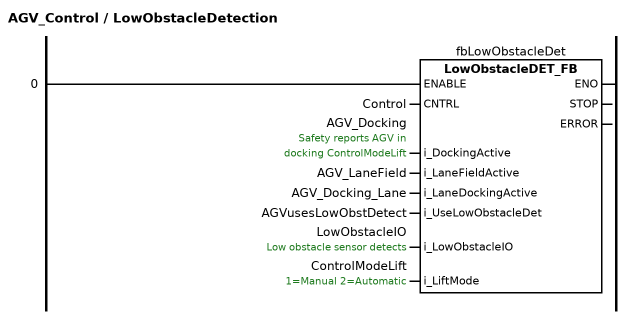
(* Rung 0 *)
fbLowObstacleDet(ENABLE := TRUE, CNTRL := Control, i_DockingActive := AGV_Docking, i_LaneFieldActive := AGV_LaneField, i_LaneDockingActive := AGV_Docking_Lane, i_UseLowObstacleDet := AGVusesLowObstDetect, i_LowObstacleIO := LowObstacleIO, i_LiftMode := ControlModeLift);

(* Section ActuatorLogic: ladder, written here as Structured Text *)

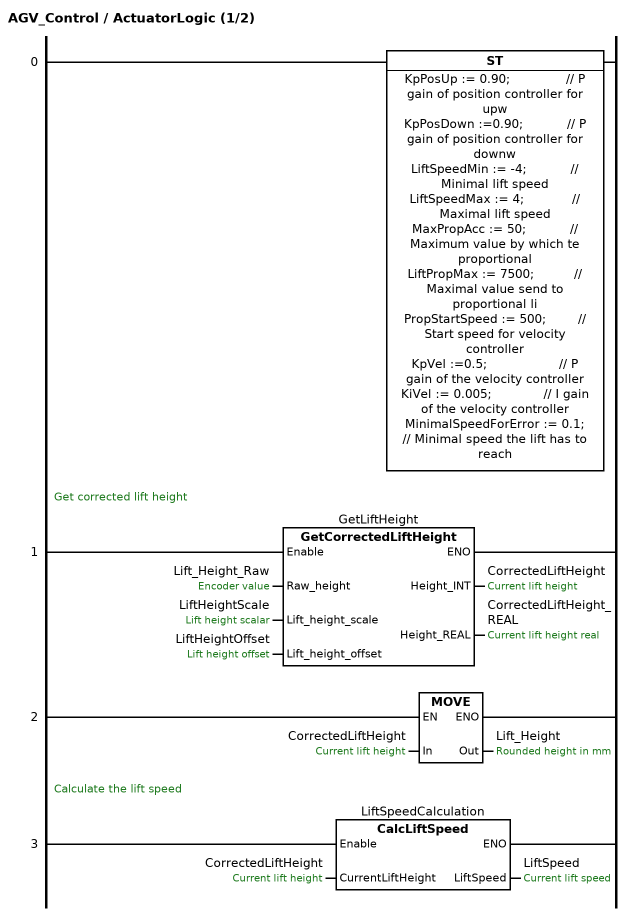
(* Rung 0 *)
KpPosUp := 0.90;							// P gain of position controller for upwards movement
KpPosDown :=0.90;						// P gain of position controller for downwards movement 
LiftSpeedMin := -4;						// Minimal lift speed
LiftSpeedMax := 4;						// Maximal lift speed
MaxPropAcc := 50;						// Maximum value by which te proportional speed is increased/decreased per cycle  
LiftPropMax := 7500;					// Maximal value send to proportional lift control
PropStartSpeed := 500;				// Start speed for velocity controller
KpVel :=0.5;									// P gain of the velocity controller
KiVel := 0.005;							// I gain of the velocity controller
MinimalSpeedForError := 0.1;		// Minimal speed the lift has to reach when the proportional speed is max. Otherwise the speed controller will give an error
(* Rung 1: Get corrected lift height *)
GetLiftHeight(Enable := TRUE, Raw_height := Lift_Height_Raw, Lift_height_scale := LiftHeightScale, Lift_height_offset := LiftHeightOffset, Height_INT => CorrectedLiftHeight, Height_REAL => CorrectedLiftHeight_REAL);
(* Rung 2 *)
Lift_Height := CorrectedLiftHeight;
(* Rung 3: Calculate the lift speed *)
LiftSpeedCalculation(Enable := TRUE, CurrentLiftHeight := CorrectedLiftHeight, LiftSpeed => LiftSpeed);

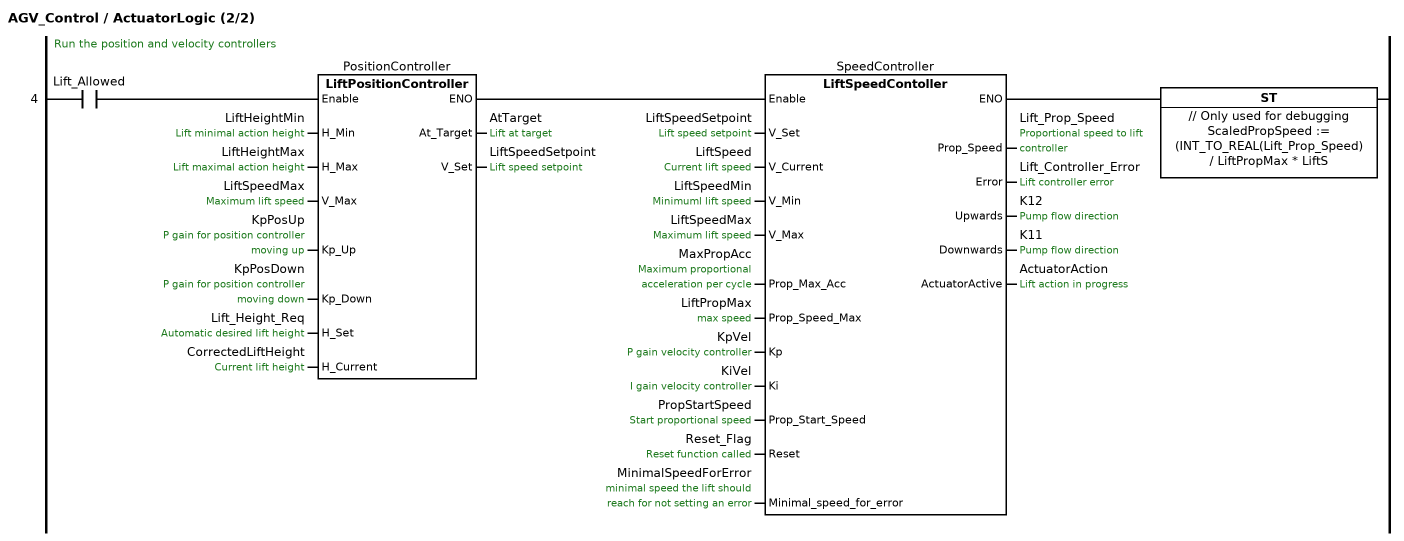
(* Rung 4: Run the position and velocity controllers *)
PositionController(Enable := Lift_Allowed, H_Min := LiftHeightMin, H_Max := LiftHeightMax, V_Max := LiftSpeedMax, Kp_Up := KpPosUp, Kp_Down := KpPosDown, H_Set := Lift_Height_Req, H_Current := CorrectedLiftHeight, At_Target => AtTarget, V_Set => LiftSpeedSetpoint);
SpeedController(Enable := PositionController.ENO, V_Set := LiftSpeedSetpoint, V_Current := LiftSpeed, V_Min := LiftSpeedMin, V_Max := LiftSpeedMax, Prop_Max_Acc := MaxPropAcc, Prop_Speed_Max := LiftPropMax, Kp := KpVel, Ki := KiVel, Prop_Start_Speed := PropStartSpeed, Reset := Reset_Flag, Minimal_speed_for_error := MinimalSpeedForError, Prop_Speed => Lift_Prop_Speed, Error => Lift_Controller_Error, Upwards => K12, Downwards => K11, ActuatorActive => ActuatorAction);
IF SpeedController.ENO THEN
    // Only used for debugging
    ScaledPropSpeed := (INT_TO_REAL(Lift_Prop_Speed) / LiftPropMax * LiftSpeedMax);
END_IF;

(* Section ActuatorControl: ladder, written here as Structured Text *)

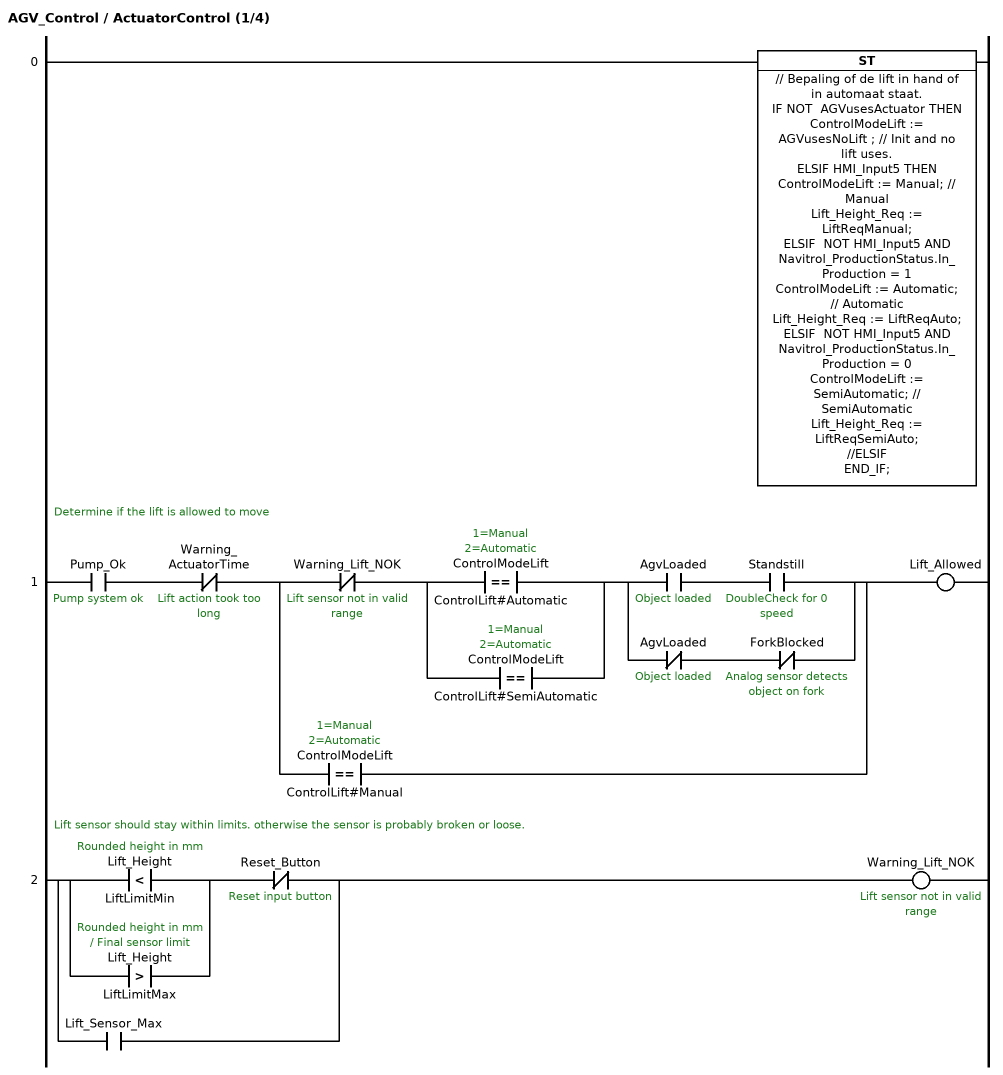
(* Rung 0 *)
// Bepaling of de lift in hand of in automaat staat.

IF NOT  AGVusesActuator THEN
	ControlModeLift := AGVusesNoLift ; // Init and no lift uses.
ELSIF HMI_Input5 THEN
	ControlModeLift := Manual; // Manual
	Lift_Height_Req := LiftReqManual;
ELSIF  NOT HMI_Input5 AND Navitrol_ProductionStatus.In_Production = 1 THEN
	ControlModeLift := Automatic; // Automatic
	  Lift_Height_Req := LiftReqAuto;
ELSIF  NOT HMI_Input5 AND Navitrol_ProductionStatus.In_Production = 0 THEN
	ControlModeLift := SemiAutomatic; // SemiAutomatic
	  Lift_Height_Req := LiftReqSemiAuto;	  
//ELSIF
END_IF;
(* Rung 1: Determine if the lift is allowed to move *)
Lift_Allowed := Pump_Ok AND NOT Warning_ActuatorTime AND ((NOT Warning_Lift_NOK AND ((ControlModeLift = ControlLift#Automatic) OR (ControlModeLift = ControlLift#SemiAutomatic)) AND ((AgvLoaded AND Standstill) OR (NOT AgvLoaded AND NOT ForkBlocked))) OR (ControlModeLift = ControlLift#Manual));
(* Rung 2: Lift sensor should stay within limits. otherwise the sensor is probably broken or loose. *)
Warning_Lift_NOK := (((Lift_Height < LiftLimitMin) OR (Lift_Height > LiftLimitMax)) AND NOT Reset_Button) OR Lift_Sensor_Max;

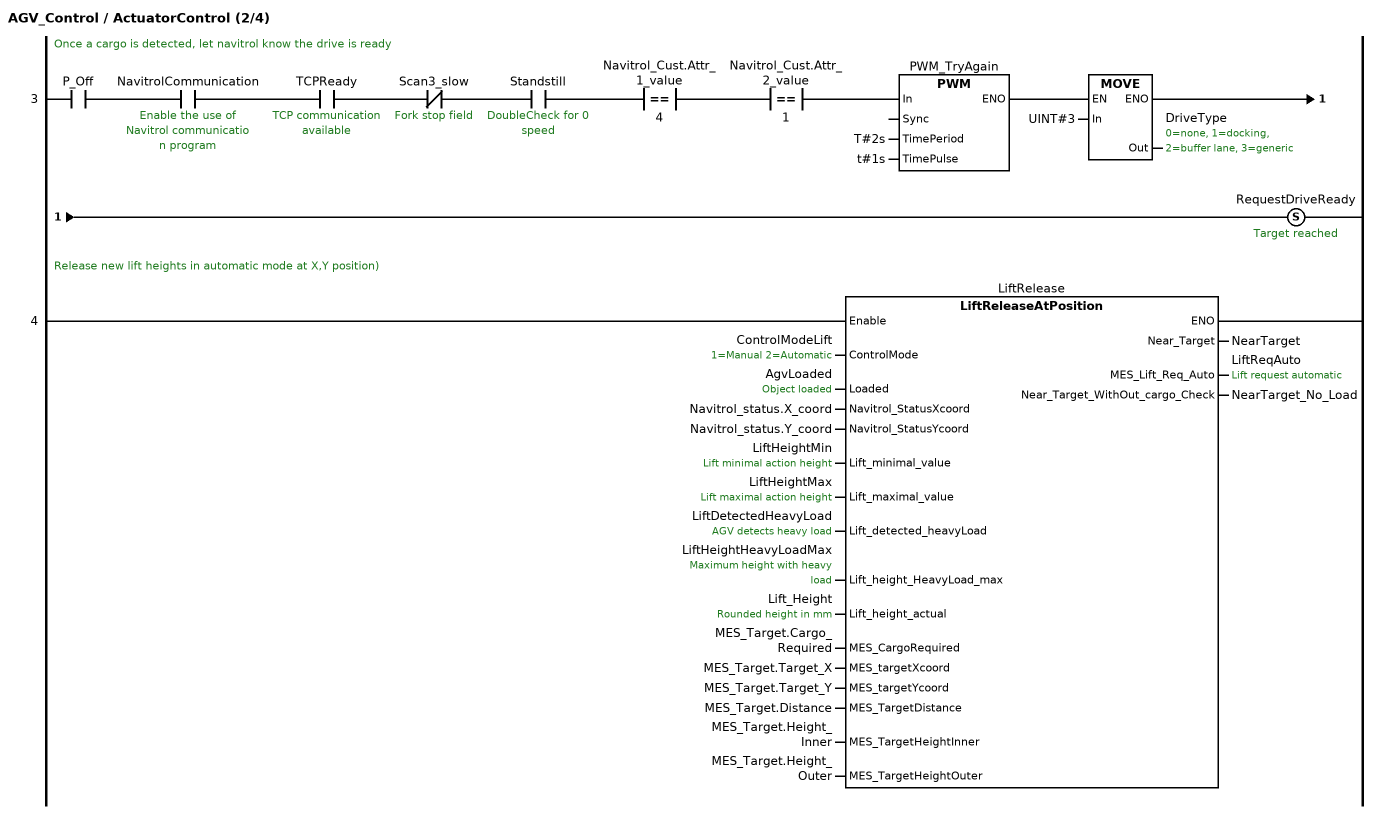
(* Rung 3: Once a cargo is detected, let navitrol know the drive is ready *)
PWM_TryAgain(In := P_Off AND NavitrolCommunication AND TCPReady AND NOT Scan3_slow AND Standstill AND (Navitrol_Cust.Attr_1_value = 4) AND (Navitrol_Cust.Attr_2_value = 1), TimePeriod := T#2s, TimePulse := t#1s);
IF PWM_TryAgain.ENO THEN
    DriveType := UINT#3;
    RequestDriveReady := TRUE;
END_IF;
(* Rung 4: Release new lift heights in automatic mode at X,Y position) *)
LiftRelease(Enable := TRUE, ControlMode := ControlModeLift, Loaded := AgvLoaded, Navitrol_StatusXcoord := Navitrol_status.X_coord, Navitrol_StatusYcoord := Navitrol_status.Y_coord, Lift_minimal_value := LiftHeightMin, Lift_maximal_value := LiftHeightMax, Lift_detected_heavyLoad := LiftDetectedHeavyLoad, Lift_height_HeavyLoad_max := LiftHeightHeavyLoadMax, Lift_height_actual := Lift_Height, MES_CargoRequired := MES_Target.Cargo_Required, MES_targetXcoord := MES_Target.Target_X, MES_targetYcoord := MES_Target.Target_Y, MES_TargetDistance := MES_Target.Distance, MES_TargetHeightInner := MES_Target.Height_Inner, MES_TargetHeightOuter := MES_Target.Height_Outer, Near_Target => NearTarget, MES_Lift_Req_Auto => LiftReqAuto, Near_Target_WithOut_cargo_Check => NearTarget_No_Load);

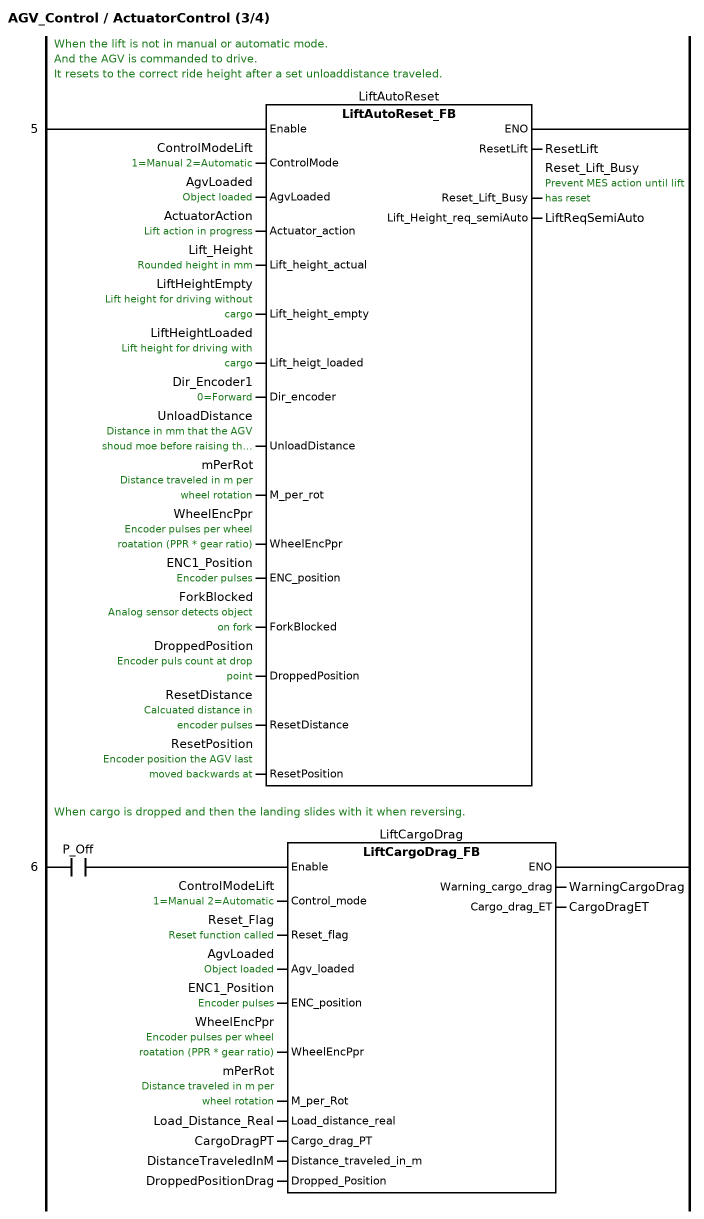
(* Rung 5: When the lift is not in manual or automatic mode. / And the AGV is commanded to drive. / It resets to the correct ride height after a set unloaddistance traveled. *)
LiftAutoReset(Enable := TRUE, ControlMode := ControlModeLift, AgvLoaded := AgvLoaded, Actuator_action := ActuatorAction, Lift_height_actual := Lift_Height, Lift_height_empty := LiftHeightEmpty, Lift_heigt_loaded := LiftHeightLoaded, Dir_encoder := Dir_Encoder1, UnloadDistance := UnloadDistance, M_per_rot := mPerRot, WheelEncPpr := WheelEncPpr, ENC_position := ENC1_Position, ForkBlocked := ForkBlocked, DroppedPosition := DroppedPosition, ResetDistance := ResetDistance, ResetPosition := ResetPosition, ResetLift => ResetLift, Reset_Lift_Busy => Reset_Lift_Busy, Lift_Height_req_semiAuto => LiftReqSemiAuto);
(* Rung 6: When cargo is dropped and then the landing slides with it when reversing. *)
LiftCargoDrag(Enable := P_Off, Control_mode := ControlModeLift, Reset_flag := Reset_Flag, Agv_loaded := AgvLoaded, ENC_position := ENC1_Position, WheelEncPpr := WheelEncPpr, M_per_Rot := mPerRot, Load_distance_real := Load_Distance_Real, Cargo_drag_PT := CargoDragPT, Distance_traveled_in_m := DistanceTraveledInM, Dropped_Position := DroppedPositionDrag, Warning_cargo_drag => WarningCargoDrag, Cargo_drag_ET => CargoDragET);

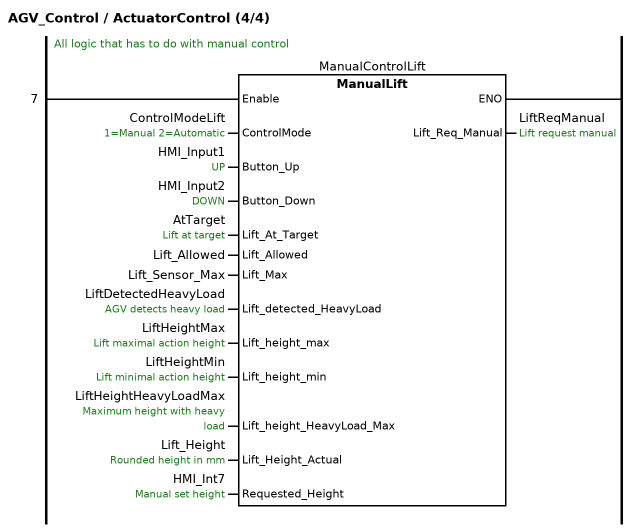
(* Rung 7: All logic that has to do with manual control *)
ManualControlLift(Enable := TRUE, ControlMode := ControlModeLift, Button_Up := HMI_Input1, Button_Down := HMI_Input2, Lift_At_Target := AtTarget, Lift_Allowed := Lift_Allowed, Lift_Max := Lift_Sensor_Max, Lift_detected_HeavyLoad := LiftDetectedHeavyLoad, Lift_height_max := LiftHeightMax, Lift_height_min := LiftHeightMin, Lift_height_HeavyLoad_Max := LiftHeightHeavyLoadMax, Lift_Height_Actual := Lift_Height, Requested_Height := HMI_Int7, Lift_Req_Manual => LiftReqManual);

(* Section LoadDetection: ladder, written here as Structured Text *)

